FUNCTION_BLOCK _BIT_UsingMockStructure_TestSuite EXTENDS TcUnit.FB_TestSuite
VAR
END_VAR

TestAddress();
TestClearReference();
TestClone();
TestTypeNameReturnsExpected();
TestMakeReferenceToFollowsReference();
TestMakeReferenceToUpdatesReference();
TestSize();
TestValueReturnsExpectedAfterChange();
TestSerializeTypeWith();
TestSerializeWith();
TestTryDeserializeFrom();
TestTryMakeReferenceToFollowsReference();
TestTryMakeReferenceToUpdatesReference();

METHOD PUBLIC TestAddress
VAR
    _type : _MyStruct;
    notExpected : PVOID := 0;
    actual : PVOID;
END_VAR
TEST('TestAddress');

actual := _type.MyBit.Address;

AssertFalse(
    Condition := (notExpected = actual),
    Message := 'Type did not return a valid address.'
);

TEST_FINISHED();
END_METHOD

METHOD PUBLIC TestClearReference
VAR
    _type : _MyStruct;
	target : MyStruct;
    expected : BOOL := FALSE;
    actual : BOOL;
END_VAR
TEST('TestClearReference');

_type.MakeReferenceTo(target);
_type.ClearReference();
target.MyBit := TRUE;

actual := _type.MyBit.Value;

AssertEquals(
    Expected := expected,
    Actual := actual,
    Message := 'Value incorrectly followed target change'
);

TEST_FINISHED();
END_METHOD

METHOD PUBLIC TestClone
VAR
    _type : _MyStruct;
	clone : I_Datatype;
	isValidClone : BOOL;
	compareResult : DINT;
END_VAR
TEST('TestClone');

clone := _type.Clone();

isValidClone := clone <> 0;

IF isValidClone THEN
	compareResult := memcmp(_type.Address, clone.Address, clone.Size);
END_IF

AssertTrue(
	Condition := isValidClone,
	Message := 'Clone did not produce a clone'
);

clone.Dispose();

TEST_FINISHED();
END_METHOD

METHOD PUBLIC TestMakeReferenceToFollowsReference
VAR
    _type : _MyStruct;
	target : MyStruct;
    expected : BOOL := TRUE;
    actual : BOOL;
END_VAR
TEST('TestMakeReferenceToFollowsReference');

_type.MakeReferenceTo(target);
target.MyBit := TRUE;

actual := _type.MyBit.Value;

AssertEquals(
    Expected := expected,
    Actual := actual,
    Message := 'Value did not follow target change'
);

TEST_FINISHED();
END_METHOD

METHOD PUBLIC TestMakeReferenceToUpdatesReference
VAR
    _type : _MyStruct;
	target : MyStruct;
    expected : BOOL := TRUE;
    actual : BOOL;
END_VAR
TEST('TestMakeReferenceToUpdatesReference');

_type.MakeReferenceTo(target);
_type.MyBit.Value:= TRUE;

actual := target.MyBit;

AssertEquals(
    Expected := expected,
    Actual := actual,
    Message := 'Value did not update target'
);

TEST_FINISHED();
END_METHOD

METHOD PUBLIC TestSerializeTypeWith
VAR
    _type : _MyStruct;
    serializer : JsonSerializer;
    expected : STRING := '{"typeName":"BIT"}';
    actual : STRING(500);
END_VAR
TEST('TestSerializeTypeWith');

serializer.Reset();
_type.MyBit.SerializeTypeWith(serializer);
serializer.TryGetSerializedData(ADR(actual), SIZEOF(actual));

AssertEquals_STRING(
    Expected := expected,
    Actual := actual,
    Message := 'Serialization of type did not return correct string.'
);

TEST_FINISHED();
END_METHOD

METHOD PUBLIC TestSerializeWith
VAR
    _type : _MyStruct;
    serializer : JsonSerializer;
    expected : STRING := 'true';
    actual : STRING(500);
END_VAR
TEST('TestSerializeWith');

serializer.Reset();
_type.MyBit.Value := true;
_type.MyBit.SerializeWith(serializer);
serializer.TryGetSerializedData(ADR(actual), SIZEOF(actual));

AssertEquals_STRING(
    Expected := expected,
    Actual := actual,
    Message := 'Serialization of type data did not return correct string.'
);

TEST_FINISHED();
END_METHOD

METHOD PUBLIC TestSize
VAR
    _type : _MyStruct;
    expected : UDINT := SIZEOF(MyStruct.MyBit);
    actual : UDINT;
END_VAR
TEST('TestSize');

actual := _type.MyBit.Size;

AssertEquals_UDINT(
    Expected := Expected,
    Actual := actual,
    Message := 'Type did not return the correct size.'
);

TEST_FINISHED();
END_METHOD

METHOD PUBLIC TestTryDeserializeFrom
VAR
    deserializer : JsonDeserializer;
    feedback : DeserializerFeedback;
    json : STRING := 'true';
    _type : _MyStruct;
    expected : BOOL := TRUE;
    actual : BOOL;
 END_VAR
TEST('TestTryDeserializeFrom');

deserializer.Reset();
deserializer.TryLoad(json);
_type.MyBit.TryDeserializeFrom(Deserializer, Feedback);

actual := _type.MyBit.Value;

AssertEquals(
    Expected := expected,
    Actual := actual,
    Message := 'Type did not deserialize correctly.'
);

TEST_FINISHED();
END_METHOD

METHOD PUBLIC TestTryMakeReferenceToFollowsReference
VAR
    _type : _MyStruct;
	target : _MyStruct;
    expected : BOOL := TRUE;
    actual : BOOL;
END_VAR
TEST('TestTryMakeReferenceToFollowsReference');

_type.TryMakeReferenceTo(target);
target.MyBit.Value := TRUE;

actual := _type.MyBit.Value;

AssertEquals(
    Expected := expected,
    Actual := actual,
    Message := 'Value did not follow target change'
);

TEST_FINISHED();
END_METHOD

METHOD PUBLIC TestTryMakeReferenceToUpdatesReference
VAR
    _type : _MyStruct;
	target : _MyStruct;
    expected : BOOL := TRUE;
    actual : BOOL;
END_VAR
TEST('TestTryMakeReferenceToUpdatesReference');

_type.TryMakeReferenceTo(target);
_type.MyBit.Value := TRUE;

actual := target.MyBit.Value;

AssertEquals(
    Expected := expected,
    Actual := actual,
    Message := 'Value did not update target'
);

TEST_FINISHED();
END_METHOD

METHOD PUBLIC TestTypeNameReturnsExpected
VAR
    _type : _MyStruct;
    expected : STRING := 'BIT';
    actual : STRING;
END_VAR
TEST('TestTypeNameReturnsExpected');

actual := _type.MyBit.TypeName;

AssertEquals_STRING(
    Expected := expected,
    Actual := actual,
    Message := 'Type did not return correct iec type.'
);

TEST_FINISHED();
END_METHOD

METHOD PUBLIC TestValueReturnsExpectedAfterChange
VAR
    _type : _MyStruct;
    expected : BOOL := FALSE;
    actual : BOOL;
END_VAR
TEST('TestValueReturnsExpectedAfterChange');

_type.MyBit.Value := FALSE;

actual := _type.MyBit.Value;

AssertEquals(
    Expected := expected,
    Actual := actual,
    Message := 'Expected value not returned after change.'
);

TEST_FINISHED();
END_METHOD

END_FUNCTION_BLOCK

(* stored: Version 1.1.0.1, ProductVersion 3.1.4024.12
   POU _BIT_UsingMockStructure_TestSuite: Id {e587821c-05b3-4279-bb93-dc39350e8beb}, SpecialFunc None
   Method TestAddress: Id {abd70174-c3d3-4946-a640-0088574c99eb}
   Method TestClearReference: Id {82c51a18-1517-4c59-879d-17c6596f4729}
   Method TestClone: Id {fadd0e7c-1103-4203-8b59-14a5dc432fad}
   Method TestMakeReferenceToFollowsReference: Id {8cd47f7f-4e3a-474c-89b0-efcc6dcf273c}
   Method TestMakeReferenceToUpdatesReference: Id {8de12234-4f9b-4653-a8ec-fd16a646d023}
   Method TestSerializeTypeWith: Id {cf8cb0bc-35c3-4ece-b7f2-70b5fb4c8655}
   Method TestSerializeWith: Id {d6281bf1-8458-4a11-9bd9-a3f6bad0d294}
   Method TestSize: Id {e0bc1320-b58e-4bdd-a457-a9c62ad50cd7}
   Method TestTryDeserializeFrom: Id {fabd89c8-7514-4393-a331-949e263848dc}
   Method TestTryMakeReferenceToFollowsReference: Id {ba5389ca-0bce-4fb2-a92d-60c9000e2103}
   Method TestTryMakeReferenceToUpdatesReference: Id {6cf47bb7-c605-4b08-a262-886dd2e2a4b9}
   Method TestTypeNameReturnsExpected: Id {12d35620-8364-4d20-ae45-d75516e09d1e}
   Method TestValueReturnsExpectedAfterChange: Id {c8bfaca2-440b-4645-96bb-d16a07aeb8e9} *)
